PROGRAM torqueInput
VAR
	

	frequency : LREAL :=0 ;
	bias : LREAL :=0.4;
	duration: LREAL := 1000;
	torqueInput: REAL:= 0.05;
	torqueStarter : BOOL:= FALSE;
	state : INT := 10;	
	counter : LREAL := 0;
	f0 :LREAL	:=0;
	f1 :LREAL:=100;
	T : LREAL ;
	
	x: LREAL;
	
	
	trial: INT := 0;
END_VAR

CASE state OF
	
10 :
	
	IF MAIN.dummy = 0 AND torqueStarter THEN
		state := 20;
	ELSIF MAIN.dummy = 1 AND torqueStarter THEN
		state := 30;
	END_IF
 
	
20 :
IF 	torqueStarter THEN
	counter := counter +1;
	IF counter < duration THEN
		T :=duration/1000.0;
		frequency := f0 + counter/1000.0 *(f1-f0)/T;	
		//link.torqueOfsetX := REAL_TO_INT(torqueInput*(1000/2.37));
		x:=SIN(2*pi*((f0*counter/1000)+((f1-f0)/(2*T)*(EXPT(counter/1000,2)))));
			IF MAIN.opertionModeRead=10 THEN
		//link.torqueOfsetX := LREAL_TO_INT(torqueInput*(1000/2.37)*x);
			link.torqueX := LREAL_TO_INT((torqueInput*1000/2.37)*(x+bias/(torqueInput)));
			
			ELSIF MAIN.opertionModeRead=9 THEN				
			link.torqueOfsetX := LREAL_TO_INT(torqueInput*(1000/2.37)*x);
			END_IF
	ELSE
		link.torqueX := 0;
		link.torqueOfsetX := 0;
		torqueStarter := FALSE;
		counter := 0;
		state := 60;
		
	END_IF
ELSE
	link.torqueOfsetX := 0;
END_IF
	
30 :
IF 	torqueStarter THEN
	counter := counter +1;
	IF counter < duration THEN
		T :=duration/1000.0;
		frequency := f0 + counter/1000.0 *(f1-f0)/T;	
		//link.torqueOfsetY := REAL_TO_INT(torqueInput*(1000/2.37));
		x:=SIN(2*pi*((f0*counter/1000)+((f1-f0)/(2*T)*(EXPT(counter/1000,2)))));
			IF MAIN.opertionModeRead=10 THEN
		//link.torqueOfsetY := LREAL_TO_INT(torqueInput*(1000/2.37)*x);
			link.torqueY := LREAL_TO_INT((torqueInput*1000/2.37)*(x+bias/(torqueInput)));
			
			ELSIF MAIN.opertionModeRead=9 THEN				
			link.torqueOfsetY := LREAL_TO_INT(torqueInput*(1000/2.37)*x);
			END_IF
	ELSE
		link.torqueY := 0;
		link.torqueOfsetY := 0;
		torqueStarter := FALSE;
		counter := 0;
		state := 60;
		
	END_IF
ELSE
	link.torqueOfsetY := 0;
END_IF
60 :
	torqueStarter:=FALSE;
	state :=10;
	counter := 0;
			
	
END_CASE

END_PROGRAM

(* stored: Version 1.1.0.1, ProductVersion 3.1.4024.9
   POU torqueInput: Id {839c653f-4f0b-4e68-9f1b-243e78656ff8}, SpecialFunc None *)
